(* IEC 61131-3 sources: Industry-PLC-LLM/data/PLCBEAD_repo/PLCBEAD_PLCEmbed-main/PLC-BEAD/Source/GEB/TRUNC_UDINT, 1 file *)

(* ---- TRUNC_UDINT.ST ---- *)
FUNCTION TRUNC_UDINT:UDINT
	VAR_INPUT
		IN :	REAL;
	END_VAR
	TRUNC_UDINT := INT_TO_UDINT(TRUNC(IN));
END_FUNCTION

PROGRAM program0
	VAR
		LocalVar0 : REAL;
		LocalOUT  : UDINT;
	END_VAR
		LocalOUT := TRUNC_UDINT(LocalVar0);
END_PROGRAM
